FUNCTION_BLOCK EL2522
VAR
	{attribute addProperty Name "WcState"}
	_wcState : WcStateInputToggle;
	{attribute addProperty Name "Info data"}
	_infoData : InfoDataAds;
	_io : EL2522_Data;
END_VAR

PROPERTY IO : REFERENCE TO EL2522_Data
GET
IO REF= _io;
END_GET
END_PROPERTY

PROPERTY WcState : REFERENCE TO WcStateInputToggle
GET
WcState REF= _wcState;
END_GET
END_PROPERTY

END_FUNCTION_BLOCK

(* stored: Version 1.1.0.1, ProductVersion 3.1.4024.9
   POU EL2522: Id {c36636ae-d96a-0712-2956-a6cdc1663e4e}, SpecialFunc None
   Property IO: Id {55d2c521-4432-068d-0c10-c5aed2ff8d7f}
   Get Get: Id {c810faa5-59f7-098d-0735-9ad19451cbf7}
   Property WcState: Id {e7dc9f8e-f6ac-07b6-13c2-415419023dec}
   Get Get: Id {3c4e7495-c214-026a-29c5-9fb0680e0ab9} *)
